TYPE ST_AxisStructRemote :
STRUCT
    stControl: ST_AxisControl;
    stStatus: ST_AxisStatus;
    stConfig: ST_AxisConfig;
    stError: ST_AxisError;
    stInputs: ST_AxisInputs;
    stDescription: ST_AxisDescription;
	stHomingConfig : ST_AxisHomingConfig;
    //The NC axis link to the hardware that is controlling
END_STRUCT
END_TYPE

(* stored: Version 1.1.0.1, ProductVersion 3.1.4026.18
   DUT ST_AxisStructRemote: Id {10376df0-1410-4dc6-821f-abcb6dadeb70} *)
